{attribute addProperty BoxType "KL2751"}
{attribute addProperty Id "Channel_1Channel_B0A8062F00"}
{attribute addProperty CRC "2809087995"}
{attribute addProperty SizeInBites "0"}
{attribute addProperty SizeInBytes "0"}
TYPE KL2751_A76F47FB :
STRUCT
	{attribute addProperty Name "Channel_1"}
	Channel_1 : Channel_B0A8062F;
END_STRUCT
END_TYPE

(* stored: Version 1.2.0.0, ProductVersion 3.1.4024.9
   DUT KL2751_A76F47FB: Id {52569ad2-37f6-473e-a112-04ec94f95260} *)
